Yaskawa INFORM job: OK_R2_O5(90,-90)OKKR_ZJEBANY.JBI

/JOB
//NAME OK_R2_O5(90,-90)OKKR_ZJEBANY
///FOLDERNAME X4
//POS
///NPOS 29,29,29,2,0,0
///TOOL 0
///POSTYPE PULSE
///PULSE
C00000=-7951,67339,-33033,-50895,88548,73848
C00001=-40954,103923,-11144,-49051,91600,71477
C00002=-115720,106175,19532,-41458,83183,72327
C00003=-120665,117566,37019,-42317,94737,69911
C00004=-120666,119569,43109,-42133,92694,70745
C00005=-120665,115469,38682,-42169,93159,70556
C00006=-120665,113738,38399,-42128,92623,70776
C00007=-120665,114622,38535,-42149,92900,70661
C00008=-121662,114644,38564,-41741,92507,70454
C00009=-120665,114622,38535,-42149,92900,70661
C00010=-117243,119756,39975,-43676,95543,70809
C00011=-117243,132866,44667,-44105,98363,69579
C00012=-120664,101755,21867,-38342,86132,69722
C00013=-120677,101990,25493,-38404,84454,70316
C00014=-120813,97941,21567,-38321,84674,70193
C00015=-120666,109345,35326,-38530,82658,70965
C00016=-120023,108618,35688,-38881,82424,71277
C00017=-120802,102796,27095,-39996,85988,71578
C00018=-120813,101468,24288,-39954,88273,70716
C00019=-120826,101479,24385,-39948,88227,70729
C00020=-120788,112192,36071,-40057,91666,69443
C00021=-120799,113296,36248,-40398,95871,67841
C00022=-120780,114304,36424,-38898,97622,65567
C00023=-120791,114701,36502,-39256,99878,64724
C00024=-120667,115659,36710,-39351,100209,64643
C00025=-120667,118516,37423,-39501,101014,64338
C00026=-115974,119000,37607,-41692,79652,73657
C00027=-46054,109823,-1861,-45657,88406,71781
C00028=-10422,67877,-32326,-49333,87682,73596
BC00000=135837,674709,1075175
BC00001=135837,677506,1075175
BC00002=135837,682951,1075175
BC00003=143646,674422,1075175
BC00004=138011,669733,1075175
BC00005=135758,672601,1075175
BC00006=135758,672601,1075175
BC00007=135758,672601,1075175
BC00008=135758,672601,1075175
BC00009=135758,672601,1075175
BC00010=135758,672601,1075175
BC00011=135758,672601,1075175
BC00012=135878,652143,1075175
BC00013=130265,650391,1075175
BC00014=128019,653981,1075175
BC00015=128019,643159,1075175
BC00016=128019,643159,1075175
BC00017=130157,658598,1075175
BC00018=130154,664330,1075175
BC00019=130154,664330,1075175
BC00020=130132,674399,1075175
BC00021=130094,689101,1075175
BC00022=127975,692548,1075175
BC00023=127978,698669,1075175
BC00024=130224,698878,1075175
BC00025=135837,699401,1075175
BC00026=135837,668931,1075175
BC00027=135837,659487,1075175
BC00028=135837,667934,1075175
EC00000=798156,-556475
EC00001=798156,-556475
EC00002=798156,-556475
EC00003=798156,-556475
EC00004=798156,-556475
EC00005=798156,-556475
EC00006=798156,-556475
EC00007=798156,-556475
EC00008=798156,-556475
EC00009=798156,-556475
EC00010=798156,-556475
EC00011=798156,-556475
EC00012=798156,-556475
EC00013=798156,-556475
EC00014=798156,-556475
EC00015=798156,-556475
EC00016=798156,-556475
EC00017=798156,-556475
EC00018=798156,-556475
EC00019=798156,-556475
EC00020=798156,-556475
EC00021=798156,-556475
EC00022=798156,-556475
EC00023=798156,-556475
EC00024=798156,-556475
EC00025=798156,-556475
EC00026=798156,-556475
EC00027=798156,-556475
EC00028=798156,-556475
///POSTYPE BASE
///RECTAN
///RCONF 0,0,0,0,0,0,0,0,0,0,0,0,0,0,0,0,0,0,0,0,0,0,0,0
P00006=0.222,-3.123,-1.508,0.0000,0.0000,0.0000
P00021=-0.225,-6.128,-0.405,0.0000,0.0000,0.0000
//INST
///DATE 2024/02/06 15:37
///ATTR SC,RW
///GROUP1 RB1,BS1
///GROUP2 ST1
NOP
MOVJ C00000 BC00000 VJ=10.00  +MOVJ EC00000 VJ=10.00
MOVJ C00001 BC00001 VJ=10.00  +MOVJ EC00001 VJ=10.00
MOVJ C00002 BC00002 VJ=10.00  +MOVJ EC00002 VJ=0.78
'OK_r2_O5(90,-90)
'Path S1553
SFTOF3D
MOVJ C00003 BC00003 VJ=100.00  +MOVJ EC00003 VJ=100.00
MOVL C00004 BC00004 V=400.0  +MOVJ EC00004 VJ=100.00
SMOVL C00005 BC00005 V=60.0  +MOVJ EC00005
SREFP 3 C00006 BC00006  +REFP EC00006
CALL JOB:SEARCH-R1-S13D
SET P021 P006
SFTON3D P021
SMOVL C00007 BC00007 V=60.0  +MOVJ EC00007
SREFP 3 C00008 BC00008  +REFP EC00008
CALL JOB:SEARCH-R1-S13D
SET P021 P006
SFTON3D P021
SMOVL C00009 BC00009 V=60.0  +MOVJ EC00009
MOVL C00010 BC00010 V=1000.0  +MOVJ EC00010 VJ=100.00
MOVL C00011 BC00011 V=1000.0  +MOVJ EC00011 VJ=100.00
'Path W936
SFTOF3D
SFTON3D P021
MOVJ C00012 BC00012 VJ=100.00  +MOVJ EC00012 VJ=100.00
SMOVL C00013 BC00013 V=400.0  +MOVJ EC00013
SMOVL C00014 BC00014 V=100.0 PL=0  +MOVJ EC00014
SREFP 1 C00015 BC00015  +REFP EC00015
SREFP 2 C00016 BC00016  +REFP EC00016
MACRO1 MJ#(0) ARGF9
ARCON
SMOVL C00017 BC00017 V=10.0  +MOVJ EC00017
SMOVL C00018 BC00018 V=10.0  +MOVJ EC00018
SMOVC C00019 BC00019 V=10.0  +MOVJ EC00019
SMOVC C00020 BC00020 V=10.0  +MOVJ EC00020
SMOVC C00021 BC00021 V=10.0  +MOVJ EC00021
SMOVC C00022 BC00022 V=10.0  +MOVJ EC00022
SMOVC C00023 BC00023 V=10.0  +MOVJ EC00023
ARCOF
SMOVL C00024 BC00024 V=400.0  +MOVJ EC00024
SMOVL C00025 BC00025 V=1000.0  +MOVJ EC00025
SFTOF3D
MOVJ C00026 BC00026 VJ=10.00  +MOVJ EC00026 VJ=0.78
MOVJ C00027 BC00027 VJ=10.00  +MOVJ EC00027 VJ=10.00
MOVJ C00028 BC00028 VJ=10.00  +MOVJ EC00028 VJ=10.00
END
